TYPE Datalogger :
STRUCT
	
	MesAlarmCode				: WORD ; 						(* Internal Akuo Alarm Code				*)
	MesWarningCode				: WORD ; 						(* Internal Akuo Warning Code       	*)
	MesEventCode				: WORD ; 						(* Internal Akuo Event Code         	*)
	 
	MesCP_Read					: BOOL; 						(* Permanent conditions for read		*)          

	MesCP_Write					: BOOL; 						(* Permanent conditions for read		*)    
                             						
END_STRUCT
END_TYPE

(* stored: Version 1.1.0.1, ProductVersion 3.1.4024.9
   DUT Datalogger: Id {f525ee17-afe3-4201-ba09-09a174f1cd83} *)
